//----------------------------------------------------------------------------//
// More step action in the list can be inserted here, upto ab is tested:      //
//----------------------------------------------------------------------------//
r007: NOP   0; //Wrong action number
      S     #sqSequencer.Error_Fault;
      JU    k007; //Exit
_007: NOP   0; // Action error handling
      JU    k007; // Exit






NETWORK
TITLE =S007:: STEP-007:: : ACTION CODE
    //================================ ACT HEADER ============================//
    // ACTION ACTION ACTION ACTION ACTION ACTION ACTION ACTION ACTION ACTION  //
    // AUTOCODE   AUTOCODE   AUTOCODE   AUTOCODE   AUTOCODE   AUTOCODE   AUTO //
    // ACTION ACTION ACTION ACTION ACTION ACTION ACTION ACTION ACTION ACTION  //
    //------------------------------------------------------------------------//
    // //Open Mx steam supply on WFI/PS lines.
    // //
    // //Log steam opened time.
    aa07: NOP   0;

    //------------------------------------------------------------------------//
    // ACT ACT ACT ACT ACT ACT ACT ACT ACT ACT ACT ACT ACT ACT ACT ACT ACT    //
    //------------------------------------------------------------------------//
    //Set emc_water to substate FLUSH and open WFI/PS supply valve.
L "dbCONST".SEL.LIQUID.PSWFI;
T #_emc_water_medium_liquid;
L 0;
T #_emc_water_runtime;
L "dbCONST".BLK.EMC2.SUBS.FLUSH;
T #_emc_water_subs;
L "dbCONST".BLK.CMD.START;
T #_emc_water_cmd;


//Log steam opened time.
SET;
S #_log_msg_steam_open;

    //------------------------------------------------------------------------//
    // VERIFY  VERIFY VERIFY VERIFY VERIFY VERIFY VERIFY VERIFY VERIFY VERIFY //
    //------------------------------------------------------------------------//
    //Verify if emc_water changed to substate FLUSH.
A(;
L   #_emc_water_subs;
L   "dbCONST".BLK.EMC2.SUBS.FLUSH;
==I;
);
    S     #sqSequencer.STEP.ActionVerified; //Action verified

    //------------------------------------------------------------------------//
    // Action done:                                                           //
    //------------------------------------------------------------------------//
    O     #sqSequencer.STEP.ActionVerified;
    O     #smc.NO_VERIFIC;       //No verification , bypass verification code
    S     #sqSequencer.STEP.ActionFinished;






    //============================= STEP FOOTER ==============================//
    // AUTOCODE   AUTOCODE   AUTOCODE   AUTOCODE   AUTOCODE   AUTOCODE   AUTO //
    // Get Ready after action finished:                                       //
    //------------------------------------------------------------------------//
    A     #sqSequencer.STEP.ActionFinished;
    JCN   k007;

    //------------------------------------------------------------------------//
    // Reset Action finished flag, ready for next step action:                //
    //------------------------------------------------------------------------//
    R     #sqSequencer.STEP.ActionVerified;
    R     #sqSequencer.STEP.ActionFinished;

    //------------------------------------------------------------------------//
    // If ALL actions are finished:                                           //
    //------------------------------------------------------------------------//
    SET   ;
    S     #sqSequencer.STEP.Finished;
    R     #sqSequencer.STEP.Active;
    S     #sqSequencer.STEP.Done[07];

    //------------------------------------------------------------------------//
    // End Step action(s):                                                    //
    //------------------------------------------------------------------------//
    JU    k007;

//----------------------------------------------------------------------------//
// Finished Step Action(s):                                                   //
//----------------------------------------------------------------------------//
k007: NOP   0;

    A     #sqStepTimerExpired;
    S     #sqSequencer.STEP.WithError[07]; // Step error flag
    S     #sqSequencer.Error_Fault;
    R     #sqStepTimer.IN;

NETWORK
TITLE =S007:STEP-007::Begin Transition
    //------------------------------------------------------------------------//
    // Begin the transition code:                                             //
    //------------------------------------------------------------------------//
    A007: NOP   0;
    R     #sqStepTimer.IN;






    //============================= TRAN HEADER ==============================//
    // AUTOCODE   AUTOCODE   AUTOCODE   AUTOCODE   AUTOCODE   AUTOCODE   AUTO //
    // Bypass transition if manual jump:                                      //
    //------------------------------------------------------------------------//
    A     #sqSequencer.STEP.Finished;
    A     #smc.TRN_AND_JUMP;     //Manual jump is set Transition as bypassed
    JCN   COMM;              //exit

NETWORK
TITLE =S007::STEP 007:TRAN 009: Pressure check
//----------------------------------------------------------------------------//
// TRAN   TRAN   TRAN   TRAN   TRAN   TRAN   TRAN   TRAN   TRAN   TRAN   TRAN //
// TRAN   TRAN   TRAN   TRAN   TRAN   TRAN   TRAN   TRAN   TRAN   TRAN   TRAN //
//----------------------------------------------------------------------------//
// Pressure increased above PRES_STM_POS. PCx013> PRES_STM_POS
//----------------------------------------------------------------------------//
// CONDITION   CONDITION   CONDITION   CONDITION   CONDITION   CONDITION   CO //
// CONDITION   CONDITION   CONDITION   CONDITION   CONDITION   CONDITION   CO //
//----------------------------------------------------------------------------//
A(;
L 	#_emc_gas_pi_vessel_pv;
L 	#_r_pres_stm_pos;
>R;
);






    //============================= TRAN FOOTER ==============================//
    // Transition jump control:                                               //
    //------------------------------------------------------------------------//
    A     #sqSequencer.STEP.JumpCtrl;
    S     #sqSequencer.STEP.Jump;
    S     #sqSequencer.STEP.jumpDone[07];

NETWORK
TITLE =S007:t009::TRANS-v: EXIT TRANSITION AND READY THE NEXT STEP
    //------------------------------------------------------------------------//
    // Check the jump flag and jump to the next step if the transition        //
    // condition is true and has set the jump flag:                           //
    //------------------------------------------------------------------------//
    A     #sqSequencer.STEP.Jump;
    JCN   x009;

    R     #sqSequencer.STEP.Jump;
    R     #sqSequencer.STEP.Finished;

    L     08;     // Load next STEPNO to jump to if transition satisfied
    T     #sqSequencer.STEP.NumberNext; //Next Step08.

    JU    COMM;              // Transition satisfied, Exit, go to next step
x009: NOP   0;






NETWORK
TITLE =S007::STEP-007:EXIT TRANSITION:
    //========================== STEP TRANSFER ===============================//
    // Jump to the common step progression code:                              //
    //------------------------------------------------------------------------//
    JU    COMM;






NETWORK
TITLE =S008: STEP-08::UO_MX_SIP : Positive pressure.
    //================================ STEP HEADER ===========================//
    // STEP008 STEP008 STEP008 STEP008
    // AUTOCODE   AUTOCODE   AUTOCODE   AUTOCODE   AUTOCODE   AUTOCODE   AUTO //
    // STEP008 STEP008 STEP008 STEP008
    //------------------------------------------------------------------------//
    // Positive pressure has been achieved.
    // Log actual positive pressure.
    //
    // Open Mx SIP condensate drain valve and vent filter drain valve.
    //------------------------------------------------------------------------//
S008: NOP   0;

      SET;
      R     #sqSequencer.STEP.jumpDone[08];
      A     #sqSequencer.CMD.Pause; //If paused jump
      JC    COMM;

NETWORK
TITLE =S008:STEP-08:Begin Action

      A     #sqSequencer.STEP.Finished;
      JC    A008; // Exit Action code, Jump to A008 Transition code

      //----------------------------------------------------------------------//
      // Begin step Action:                                                   //
      //----------------------------------------------------------------------//
      A     #sqSequencer.STEP.Active;
      JC    L008; // Action number loaded, Jump to L008--Step Action List

      //----------------------------------------------------------------------//
      // Load Default/Initial Step action number:                             //
      //----------------------------------------------------------------------//
      S     #sqSequencer.STEP.Active;
      S     #sqStepTimer.IN;
      L     1; //First Action, Step must contain Minimum one action
      T     #sqSequencer.STEP.ActionNumber;

//----------------------------------------------------------------------------//
// Step action list.                                                          //
// aann=mini Action step number(aa) inside main step number(nn)               //
// First Action aa00, Second action ab00, Third ac00, etc.                    //
//----------------------------------------------------------------------------//
L008: NOP   0;

      L     #sqSequencer.STEP.ActionNumber;
      JL    r008; //Wrong Action number
      JU    _008; //Action error handling
       JU    aa08; //ACTION-01
JU    ab08; //ACTION-02


//----------------------------------------------------------------------------//
// More step action in the list can be inserted here, upto ab is tested:      //
//----------------------------------------------------------------------------//
r008: NOP   0; //Wrong action number
      S     #sqSequencer.Error_Fault;
      JU    k008; //Exit
_008: NOP   0; // Action error handling
      JU    k008; // Exit






NETWORK
TITLE =S008:: STEP-008:: : ACTION CODE
    //================================ ACT HEADER ============================//
    // ACTION ACTION ACTION ACTION ACTION ACTION ACTION ACTION ACTION ACTION  //
    // AUTOCODE   AUTOCODE   AUTOCODE   AUTOCODE   AUTOCODE   AUTOCODE   AUTO //
    // ACTION ACTION ACTION ACTION ACTION ACTION ACTION ACTION ACTION ACTION  //
    //------------------------------------------------------------------------//
    // //Log actual positive pressure.
    // //Open Mx SIP condensate drain valve and vent filter drain valve.
    aa08: NOP   0;

    //------------------------------------------------------------------------//
    // ACT ACT ACT ACT ACT ACT ACT ACT ACT ACT ACT ACT ACT ACT ACT ACT ACT    //
    //------------------------------------------------------------------------//
    //Log actual positive pressure.
L #_emc_gas_pi_vessel_pv;
T #_real_positive_pressure;

SET;
S #_log_real_positive_pressure;

//Start EMX4_SIP.
L "dbCONST".BLK.EMX4.SUBS.SIP;
T #_emx_drain_subs;
L "dbCONST".BLK.CMD.START;
T #_emx_drain_cmd;

// Set vessel VENT filter EM to substate SIP
L "dbCONST".BLK.EMG1.SUBS.SIP;
T #_emg_filter_subs;
L "dbCONST".BLK.CMD.START;
T #_emg_filter_cmd;

//Open gas line drain valve.
L "dbCONST".SEL.GAS.DRAIN;
T #_emc_gas_medium_gas;
L "dbCONST".BLK.CMD.RESTART;
T #_emc_gas_cmd;

    //------------------------------------------------------------------------//
    // VERIFY  VERIFY VERIFY VERIFY VERIFY VERIFY VERIFY VERIFY VERIFY VERIFY //
    //------------------------------------------------------------------------//
    A(;
L #_emx_drain_subs;
L "dbCONST".BLK.EMX4.SUBS.SIP;
==I;
);
A(;
L #_emg_filter_subs;
L "dbCONST".BLK.EMG1.SUBS.SIP;
==I;
);
A(;
L   #_emc_gas_state;
L   "dbCONST".BLK.STATE.STOPPED;
>I;
);
A(;
L   #_emc_gas_state;
L   "dbCONST".BLK.STATE.INTERLOCKED;
<I;
);

    S     #sqSequencer.STEP.ActionVerified; //Action verified

    //------------------------------------------------------------------------//
    // Action done:                                                           //
    //------------------------------------------------------------------------//
    O     #sqSequencer.STEP.ActionVerified;
    O     #smc.NO_VERIFIC;       //No verification , bypass verification code
    S     #sqSequencer.STEP.ActionFinished;






    //============================= ACT FOOTER ===============================//
    // AUTOCODE   AUTOCODE   AUTOCODE   AUTOCODE   AUTOCODE   AUTOCODE   AUTO //
    // Get Ready after action finished:                                       //
    //------------------------------------------------------------------------//
    A     #sqSequencer.STEP.ActionFinished;
    JCN   k008;

    //------------------------------------------------------------------------//
    // Reset Action finished flag, ready for next step action:                //
    //------------------------------------------------------------------------//
    R     #sqSequencer.STEP.ActionVerified;
    R     #sqSequencer.STEP.ActionFinished;

    //------------------------------------------------------------------------//
    // Load Next Step Action number:                                          //
    //------------------------------------------------------------------------//
    L     02; //Load next Action
    T     #sqSequencer.STEP.ActionNumber;






NETWORK
TITLE =S008:: STEP-008:: : ACTION CODE
    //================================ ACT HEADER ============================//
    // ACTION ACTION ACTION ACTION ACTION ACTION ACTION ACTION ACTION ACTION  //
    // AUTOCODE   AUTOCODE   AUTOCODE   AUTOCODE   AUTOCODE   AUTOCODE   AUTO //
    // ACTION ACTION ACTION ACTION ACTION ACTION ACTION ACTION ACTION ACTION  //
    //------------------------------------------------------------------------//
    // //Clear gas EM restart command
    ab08: NOP   0;

    //------------------------------------------------------------------------//
    // ACT ACT ACT ACT ACT ACT ACT ACT ACT ACT ACT ACT ACT ACT ACT ACT ACT    //
    //------------------------------------------------------------------------//
    L "dbCONST".BLK.CMD.START;
T #_emc_gas_cmd;

    //------------------------------------------------------------------------//
    // VERIFY  VERIFY VERIFY VERIFY VERIFY VERIFY VERIFY VERIFY VERIFY VERIFY //
    //------------------------------------------------------------------------//

    S     #sqSequencer.STEP.ActionVerified; //Action verified

    //------------------------------------------------------------------------//
    // Action done:                                                           //
    //------------------------------------------------------------------------//
    O     #sqSequencer.STEP.ActionVerified;
    O     #smc.NO_VERIFIC;       //No verification , bypass verification code
    S     #sqSequencer.STEP.ActionFinished;






    //============================= STEP FOOTER ==============================//
    // AUTOCODE   AUTOCODE   AUTOCODE   AUTOCODE   AUTOCODE   AUTOCODE   AUTO //
    // Get Ready after action finished:                                       //
    //------------------------------------------------------------------------//
    A     #sqSequencer.STEP.ActionFinished;
    JCN   k008;

    //------------------------------------------------------------------------//
    // Reset Action finished flag, ready for next step action:                //
    //------------------------------------------------------------------------//
    R     #sqSequencer.STEP.ActionVerified;
    R     #sqSequencer.STEP.ActionFinished;

    //------------------------------------------------------------------------//
    // If ALL actions are finished:                                           //
    //------------------------------------------------------------------------//
    SET   ;
    S     #sqSequencer.STEP.Finished;
    R     #sqSequencer.STEP.Active;
    S     #sqSequencer.STEP.Done[08];

    //------------------------------------------------------------------------//
    // End Step action(s):                                                    //
    //------------------------------------------------------------------------//
    JU    k008;

//----------------------------------------------------------------------------//
// Finished Step Action(s):                                                   //
//----------------------------------------------------------------------------//
k008: NOP   0;

    A     #sqStepTimerExpired;
    S     #sqSequencer.STEP.WithError[08]; // Step error flag
    S     #sqSequencer.Error_Fault;
    R     #sqStepTimer.IN;

NETWORK
TITLE =S008:STEP-008::Begin Transition
    //------------------------------------------------------------------------//
    // Begin the transition code:                                             //
    //------------------------------------------------------------------------//
    A008: NOP   0;
    R     #sqStepTimer.IN;






    //============================= TRAN HEADER ==============================//
    // AUTOCODE   AUTOCODE   AUTOCODE   AUTOCODE   AUTOCODE   AUTOCODE   AUTO //
    // Bypass transition if manual jump:                                      //
    //------------------------------------------------------------------------//
    A     #sqSequencer.STEP.Finished;
    A     #smc.TRN_AND_JUMP;     //Manual jump is set Transition as bypassed
    JCN   COMM;              //exit

NETWORK
TITLE =S008::STEP 008:TRAN 010: Empty Transition
//----------------------------------------------------------------------------//
// TRAN   TRAN   TRAN   TRAN   TRAN   TRAN   TRAN   TRAN   TRAN   TRAN   TRAN //
// TRAN   TRAN   TRAN   TRAN   TRAN   TRAN   TRAN   TRAN   TRAN   TRAN   TRAN //
//----------------------------------------------------------------------------//
// Empty Transition
//----------------------------------------------------------------------------//
// CONDITION   CONDITION   CONDITION   CONDITION   CONDITION   CONDITION   CO //
// CONDITION   CONDITION   CONDITION   CONDITION   CONDITION   CONDITION   CO //
//----------------------------------------------------------------------------//
A "uncondJump";






    //============================= TRAN FOOTER ==============================//
    // Transition jump control:                                               //
    //------------------------------------------------------------------------//
    A     #sqSequencer.STEP.JumpCtrl;
    S     #sqSequencer.STEP.Jump;
    S     #sqSequencer.STEP.jumpDone[08];

NETWORK
TITLE =S008:t010::TRANS-v: EXIT TRANSITION AND READY THE NEXT STEP
    //------------------------------------------------------------------------//
    // Check the jump flag and jump to the next step if the transition        //
    // condition is true and has set the jump flag:                           //
    //------------------------------------------------------------------------//
    A     #sqSequencer.STEP.Jump;
    JCN   x010;

    R     #sqSequencer.STEP.Jump;
    R     #sqSequencer.STEP.Finished;

    L     09;     // Load next STEPNO to jump to if transition satisfied
    T     #sqSequencer.STEP.NumberNext; //Next Step09.

    JU    COMM;              // Transition satisfied, Exit, go to next step
x010: NOP   0;






NETWORK
TITLE =S008::STEP-008:EXIT TRANSITION:
    //========================== STEP TRANSFER ===============================//
    // Jump to the common step progression code:                              //
    //------------------------------------------------------------------------//
    JU    COMM;






NETWORK
TITLE =S009: STEP-09::UO_MX_SIP : Wait for free steaming timer
    //================================ STEP HEADER ===========================//
    // STEP009 STEP009 STEP009 STEP009
    // AUTOCODE   AUTOCODE   AUTOCODE   AUTOCODE   AUTOCODE   AUTOCODE   AUTO //
    // STEP009 STEP009 STEP009 STEP009
    //------------------------------------------------------------------------//
    // Start timer TIME_STM_DRAIN_Mx
    //------------------------------------------------------------------------//
S009: NOP   0;

      SET;
      R     #sqSequencer.STEP.jumpDone[09];
      A     #sqSequencer.CMD.Pause; //If paused jump
      JC    COMM;

NETWORK
TITLE =S009:STEP-09:Begin Action

      A     #sqSequencer.STEP.Finished;
      JC    A009; // Exit Action code, Jump to A009 Transition code

      //----------------------------------------------------------------------//
      // Begin step Action:                                                   //
      //----------------------------------------------------------------------//
      A     #sqSequencer.STEP.Active;
      JC    L009; // Action number loaded, Jump to L009--Step Action List

      //----------------------------------------------------------------------//
      // Load Default/Initial Step action number:                             //
      //----------------------------------------------------------------------//
      S     #sqSequencer.STEP.Active;
      S     #sqStepTimer.IN;
      L     1; //First Action, Step must contain Minimum one action
      T     #sqSequencer.STEP.ActionNumber;

//----------------------------------------------------------------------------//
// Step action list.                                                          //
// aann=mini Action step number(aa) inside main step number(nn)               //
// First Action aa00, Second action ab00, Third ac00, etc.                    //
//----------------------------------------------------------------------------//
L009: NOP   0;

      L     #sqSequencer.STEP.ActionNumber;
      JL    r009; //Wrong Action number
      JU    _009; //Action error handling
       JU    aa09; //ACTION-01


//----------------------------------------------------------------------------//
// More step action in the list can be inserted here, upto ab is tested:      //
//----------------------------------------------------------------------------//
r009: NOP   0; //Wrong action number
      S     #sqSequencer.Error_Fault;
      JU    k009; //Exit
_009: NOP   0; // Action error handling
      JU    k009; // Exit






NETWORK
TITLE =S009:: STEP-009:: : ACTION CODE
    //================================ ACT HEADER ============================//
    // ACTION ACTION ACTION ACTION ACTION ACTION ACTION ACTION ACTION ACTION  //
    // AUTOCODE   AUTOCODE   AUTOCODE   AUTOCODE   AUTOCODE   AUTOCODE   AUTO //
    // ACTION ACTION ACTION ACTION ACTION ACTION ACTION ACTION ACTION ACTION  //
    //------------------------------------------------------------------------//
    // //Start timer TIME_STM_DRAIN_Mx
    aa09: NOP   0;

    //------------------------------------------------------------------------//
    // ACT ACT ACT ACT ACT ACT ACT ACT ACT ACT ACT ACT ACT ACT ACT ACT ACT    //
    //------------------------------------------------------------------------//
    //Start Timer for steaming
A #SQ_TIMER.Q;
R #sqSeqTimerStart;

AN #SQ_TIMER.Q;
S #sqSeqTimerStart;
L #_r_time_stm_drain_mx;
L 1000;
*I;
T #SQ_TIMER.PT;

    //------------------------------------------------------------------------//
    // VERIFY  VERIFY VERIFY VERIFY VERIFY VERIFY VERIFY VERIFY VERIFY VERIFY //
    //------------------------------------------------------------------------//
    A #sqSeqTimerStart;
    S     #sqSequencer.STEP.ActionVerified; //Action verified

    //------------------------------------------------------------------------//
    // Action done:                                                           //
    //------------------------------------------------------------------------//
    O     #sqSequencer.STEP.ActionVerified;
    O     #smc.NO_VERIFIC;       //No verification , bypass verification code
    S     #sqSequencer.STEP.ActionFinished;






    //============================= STEP FOOTER ==============================//
    // AUTOCODE   AUTOCODE   AUTOCODE   AUTOCODE   AUTOCODE   AUTOCODE   AUTO //
    // Get Ready after action finished:                                       //
    //------------------------------------------------------------------------//
    A     #sqSequencer.STEP.ActionFinished;
    JCN   k009;

    //------------------------------------------------------------------------//
    // Reset Action finished flag, ready for next step action:                //
    //------------------------------------------------------------------------//
    R     #sqSequencer.STEP.ActionVerified;
    R     #sqSequencer.STEP.ActionFinished;

    //------------------------------------------------------------------------//
    // If ALL actions are finished:                                           //
    //------------------------------------------------------------------------//
    SET   ;
    S     #sqSequencer.STEP.Finished;
    R     #sqSequencer.STEP.Active;
    S     #sqSequencer.STEP.Done[09];

    //------------------------------------------------------------------------//
    // End Step action(s):                                                    //
    //------------------------------------------------------------------------//
    JU    k009;

//----------------------------------------------------------------------------//
// Finished Step Action(s):                                                   //
//----------------------------------------------------------------------------//
k009: NOP   0;

    A     #sqStepTimerExpired;
    S     #sqSequencer.STEP.WithError[09]; // Step error flag
    S     #sqSequencer.Error_Fault;
    R     #sqStepTimer.IN;

NETWORK
TITLE =S009:STEP-009::Begin Transition
    //------------------------------------------------------------------------//
    // Begin the transition code:                                             //
    //------------------------------------------------------------------------//
    A009: NOP   0;
    R     #sqStepTimer.IN;






    //============================= TRAN HEADER ==============================//
    // AUTOCODE   AUTOCODE   AUTOCODE   AUTOCODE   AUTOCODE   AUTOCODE   AUTO //
    // Bypass transition if manual jump:                                      //
    //------------------------------------------------------------------------//
    A     #sqSequencer.STEP.Finished;
    A     #smc.TRN_AND_JUMP;     //Manual jump is set Transition as bypassed
    JCN   COMM;              //exit

NETWORK
TITLE =S009::STEP 009:TRAN 011: Timer expired
//----------------------------------------------------------------------------//
// TRAN   TRAN   TRAN   TRAN   TRAN   TRAN   TRAN   TRAN   TRAN   TRAN   TRAN //
// TRAN   TRAN   TRAN   TRAN   TRAN   TRAN   TRAN   TRAN   TRAN   TRAN   TRAN //
//----------------------------------------------------------------------------//
// Timer TIME_STM_DRAIN_Mx expired?
//----------------------------------------------------------------------------//
// CONDITION   CONDITION   CONDITION   CONDITION   CONDITION   CONDITION   CO //
// CONDITION   CONDITION   CONDITION   CONDITION   CONDITION   CONDITION   CO //
//----------------------------------------------------------------------------//
A #SQ_TIMER.Q;






    //============================= TRAN FOOTER ==============================//
    // Transition jump control:                                               //
    //------------------------------------------------------------------------//
    A     #sqSequencer.STEP.JumpCtrl;
    S     #sqSequencer.STEP.Jump;
    S     #sqSequencer.STEP.jumpDone[09];

NETWORK
TITLE =S009:t011::TRANS-v: EXIT TRANSITION AND READY THE NEXT STEP
    //------------------------------------------------------------------------//
    // Check the jump flag and jump to the next step if the transition        //
    // condition is true and has set the jump flag:                           //
    //------------------------------------------------------------------------//
    A     #sqSequencer.STEP.Jump;
    JCN   x011;

    R     #sqSequencer.STEP.Jump;
    R     #sqSequencer.STEP.Finished;

    L     10;     // Load next STEPNO to jump to if transition satisfied
    T     #sqSequencer.STEP.NumberNext; //Next Step10.

    JU    COMM;              // Transition satisfied, Exit, go to next step
x011: NOP   0;






NETWORK
TITLE =S009::STEP-009:EXIT TRANSITION:
    //========================== STEP TRANSFER ===============================//
    // Jump to the common step progression code:                              //
    //------------------------------------------------------------------------//
    JU    COMM;






NETWORK
TITLE =S010: STEP-10::UO_MX_SIP : Free steam complete.
    //================================ STEP HEADER ===========================//
    // STEP010 STEP010 STEP010 STEP010
    // AUTOCODE   AUTOCODE   AUTOCODE   AUTOCODE   AUTOCODE   AUTOCODE   AUTO //
    // STEP010 STEP010 STEP010 STEP010
    //------------------------------------------------------------------------//
    // Log closed system steaming start time
    //------------------------------------------------------------------------//
S010: NOP   0;

      SET;
      R     #sqSequencer.STEP.jumpDone[10];
      A     #sqSequencer.CMD.Pause; //If paused jump
      JC    COMM;

NETWORK
TITLE =S010:STEP-10:Begin Action

      A     #sqSequencer.STEP.Finished;
      JC    A010; // Exit Action code, Jump to A010 Transition code

      //----------------------------------------------------------------------//
      // Begin step Action:                                                   //
      //----------------------------------------------------------------------//
      A     #sqSequencer.STEP.Active;
      JC    L010; // Action number loaded, Jump to L010--Step Action List

      //----------------------------------------------------------------------//
      // Load Default/Initial Step action number:                             //
      //----------------------------------------------------------------------//
      S     #sqSequencer.STEP.Active;
      S     #sqStepTimer.IN;
      L     1; //First Action, Step must contain Minimum one action
      T     #sqSequencer.STEP.ActionNumber;

//----------------------------------------------------------------------------//
// Step action list.                                                          //
// aann=mini Action step number(aa) inside main step number(nn)               //
// First Action aa00, Second action ab00, Third ac00, etc.                    //
//----------------------------------------------------------------------------//
L010: NOP   0;

      L     #sqSequencer.STEP.ActionNumber;
      JL    r010; //Wrong Action number
      JU    _010; //Action error handling
       JU    aa10; //ACTION-01
JU    ab10; //ACTION-02


//----------------------------------------------------------------------------//
// More step action in the list can be inserted here, upto ab is tested:      //
//----------------------------------------------------------------------------//
r010: NOP   0; //Wrong action number
      S     #sqSequencer.Error_Fault;
      JU    k010; //Exit
_010: NOP   0; // Action error handling
      JU    k010; // Exit






NETWORK
TITLE =S010:: STEP-010:: : ACTION CODE
    //================================ ACT HEADER ============================//
    // ACTION ACTION ACTION ACTION ACTION ACTION ACTION ACTION ACTION ACTION  //
    // AUTOCODE   AUTOCODE   AUTOCODE   AUTOCODE   AUTOCODE   AUTOCODE   AUTO //
    // ACTION ACTION ACTION ACTION ACTION ACTION ACTION ACTION ACTION ACTION  //
    //------------------------------------------------------------------------//
    // //Stop MMFLx to reset it
    aa10: NOP   0;

    //------------------------------------------------------------------------//
    // ACT ACT ACT ACT ACT ACT ACT ACT ACT ACT ACT ACT ACT ACT ACT ACT ACT    //
    //------------------------------------------------------------------------//
    L "dbCONST".BLK.CMD.STOP;
T #_emx_mmfl_cmd;

    //------------------------------------------------------------------------//
    // VERIFY  VERIFY VERIFY VERIFY VERIFY VERIFY VERIFY VERIFY VERIFY VERIFY //
    //------------------------------------------------------------------------//
    A(;
L   #_emx_mmfl_state;
L   "dbCONST".BLK.STATE.STOPPED;
==I;
);
    S     #sqSequencer.STEP.ActionVerified; //Action verified

    //------------------------------------------------------------------------//
    // Action done:                                                           //
    //------------------------------------------------------------------------//
    O     #sqSequencer.STEP.ActionVerified;
    O     #smc.NO_VERIFIC;       //No verification , bypass verification code
    S     #sqSequencer.STEP.ActionFinished;






    //============================= ACT FOOTER ===============================//
    // AUTOCODE   AUTOCODE   AUTOCODE   AUTOCODE   AUTOCODE   AUTOCODE   AUTO //
    // Get Ready after action finished:                                       //
    //------------------------------------------------------------------------//
    A     #sqSequencer.STEP.ActionFinished;
    JCN   k010;

    //------------------------------------------------------------------------//
    // Reset Action finished flag, ready for next step action:                //
    //------------------------------------------------------------------------//
    R     #sqSequencer.STEP.ActionVerified;
    R     #sqSequencer.STEP.ActionFinished;

    //------------------------------------------------------------------------//
    // Load Next Step Action number:                                          //
    //------------------------------------------------------------------------//
    L     02; //Load next Action
    T     #sqSequencer.STEP.ActionNumber;






NETWORK
TITLE =S010:: STEP-010:: : ACTION CODE
    //================================ ACT HEADER ============================//
    // ACTION ACTION ACTION ACTION ACTION ACTION ACTION ACTION ACTION ACTION  //
    // AUTOCODE   AUTOCODE   AUTOCODE   AUTOCODE   AUTOCODE   AUTOCODE   AUTO //
    // ACTION ACTION ACTION ACTION ACTION ACTION ACTION ACTION ACTION ACTION  //
    //------------------------------------------------------------------------//
    // //Log closed system start time
    // //Start pulsing MMFLx valves
    ab10: NOP   0;

    //------------------------------------------------------------------------//
    // ACT ACT ACT ACT ACT ACT ACT ACT ACT ACT ACT ACT ACT ACT ACT ACT ACT    //
    //------------------------------------------------------------------------//
    //Log closed system start time.
SET;
S #_log_msg_steam_closed;

// Set emx_mmfl to substate SIP_PULSE and start it.
L _r_time_mmflx_pulse_heat;
L 1000;
*I;
T #_emx_mmfl_opened_time;
L "dbCONST".BLK.EMX1.SUBS.SIP_PULSE;
T #_emx_mmfl_subs;
L "dbCONST".BLK.CMD.START;
T #_emx_mmfl_cmd;

    //------------------------------------------------------------------------//
    // VERIFY  VERIFY VERIFY VERIFY VERIFY VERIFY VERIFY VERIFY VERIFY VERIFY //
    //------------------------------------------------------------------------//

    S     #sqSequencer.STEP.ActionVerified; //Action verified

    //------------------------------------------------------------------------//
    // Action done:                                                           //
    //------------------------------------------------------------------------//
    O     #sqSequencer.STEP.ActionVerified;
    O     #smc.NO_VERIFIC;       //No verification , bypass verification code
    S     #sqSequencer.STEP.ActionFinished;






    //============================= STEP FOOTER ==============================//
    // AUTOCODE   AUTOCODE   AUTOCODE   AUTOCODE   AUTOCODE   AUTOCODE   AUTO //
    // Get Ready after action finished:                                       //
    //------------------------------------------------------------------------//
    A     #sqSequencer.STEP.ActionFinished;
    JCN   k010;

    //------------------------------------------------------------------------//
    // Reset Action finished flag, ready for next step action:                //
    //------------------------------------------------------------------------//
    R     #sqSequencer.STEP.ActionVerified;
    R     #sqSequencer.STEP.ActionFinished;

    //------------------------------------------------------------------------//
    // If ALL actions are finished:                                           //
    //------------------------------------------------------------------------//
    SET   ;
    S     #sqSequencer.STEP.Finished;
    R     #sqSequencer.STEP.Active;
    S     #sqSequencer.STEP.Done[10];

    //------------------------------------------------------------------------//
    // End Step action(s):                                                    //
    //------------------------------------------------------------------------//
    JU    k010;

//----------------------------------------------------------------------------//
// Finished Step Action(s):                                                   //
//----------------------------------------------------------------------------//
k010: NOP   0;

    A     #sqStepTimerExpired;
    S     #sqSequencer.STEP.WithError[10]; // Step error flag
    S     #sqSequencer.Error_Fault;
    R     #sqStepTimer.IN;

NETWORK
TITLE =S010:STEP-010::Begin Transition
    //------------------------------------------------------------------------//
    // Begin the transition code:                                             //
    //------------------------------------------------------------------------//
    A010: NOP   0;
    R     #sqStepTimer.IN;






    //============================= TRAN HEADER ==============================//
    // AUTOCODE   AUTOCODE   AUTOCODE   AUTOCODE   AUTOCODE   AUTOCODE   AUTO //
    // Bypass transition if manual jump:                                      //
    //------------------------------------------------------------------------//
    A     #sqSequencer.STEP.Finished;
    A     #smc.TRN_AND_JUMP;     //Manual jump is set Transition as bypassed
    JCN   COMM;              //exit

NETWORK
TITLE =S010::STEP 010:TRAN 012: Empty Transition
//----------------------------------------------------------------------------//
// TRAN   TRAN   TRAN   TRAN   TRAN   TRAN   TRAN   TRAN   TRAN   TRAN   TRAN //
// TRAN   TRAN   TRAN   TRAN   TRAN   TRAN   TRAN   TRAN   TRAN   TRAN   TRAN //
//----------------------------------------------------------------------------//
// Empty Transition
//----------------------------------------------------------------------------//
// CONDITION   CONDITION   CONDITION   CONDITION   CONDITION   CONDITION   CO //
// CONDITION   CONDITION   CONDITION   CONDITION   CONDITION   CONDITION   CO //
//----------------------------------------------------------------------------//
A "uncondJump";






    //============================= TRAN FOOTER ==============================//
    // Transition jump control:                                               //
    //------------------------------------------------------------------------//
    A     #sqSequencer.STEP.JumpCtrl;
    S     #sqSequencer.STEP.Jump;
    S     #sqSequencer.STEP.jumpDone[10];

NETWORK
TITLE =S010:t012::TRANS-v: EXIT TRANSITION AND READY THE NEXT STEP
    //------------------------------------------------------------------------//
    // Check the jump flag and jump to the next step if the transition        //
    // condition is true and has set the jump flag:                           //
    //------------------------------------------------------------------------//
    A     #sqSequencer.STEP.Jump;
    JCN   x012;

    R     #sqSequencer.STEP.Jump;
    R     #sqSequencer.STEP.Finished;

    L     11;     // Load next STEPNO to jump to if transition satisfied
    T     #sqSequencer.STEP.NumberNext; //Next Step11.

    JU    COMM;              // Transition satisfied, Exit, go to next step
x012: NOP   0;






NETWORK
TITLE =S010::STEP-010:EXIT TRANSITION:
    //========================== STEP TRANSFER ===============================//
    // Jump to the common step progression code:                              //
    //------------------------------------------------------------------------//
    JU    COMM;






NETWORK
TITLE =S011: STEP-11::UO_MX_SIP : SIP Started
    //================================ STEP HEADER ===========================//
    // STEP011 STEP011 STEP011 STEP011
    // AUTOCODE   AUTOCODE   AUTOCODE   AUTOCODE   AUTOCODE   AUTOCODE   AUTO //
    // STEP011 STEP011 STEP011 STEP011
    //------------------------------------------------------------------------//
    // Skip timer for SIP_ABORT if sip_timer_started=FALSE.
    //------------------------------------------------------------------------//
S011: NOP   0;

      SET;
      R     #sqSequencer.STEP.jumpDone[11];
      A     #sqSequencer.CMD.Pause; //If paused jump
      JC    COMM;

NETWORK
TITLE =S011:STEP-11:Begin Action

      A     #sqSequencer.STEP.Finished;
      JC    A011; // Exit Action code, Jump to A011 Transition code

      //----------------------------------------------------------------------//
      // Begin step Action:                                                   //
      //----------------------------------------------------------------------//
      A     #sqSequencer.STEP.Active;
      JC    L011; // Action number loaded, Jump to L011--Step Action List

      //----------------------------------------------------------------------//
      // Load Default/Initial Step action number:                             //
      //----------------------------------------------------------------------//
      S     #sqSequencer.STEP.Active;
      S     #sqStepTimer.IN;
      L     1; //First Action, Step must contain Minimum one action
      T     #sqSequencer.STEP.ActionNumber;

//----------------------------------------------------------------------------//
// Step action list.                                                          //
// aann=mini Action step number(aa) inside main step number(nn)               //
// First Action aa00, Second action ab00, Third ac00, etc.                    //
//----------------------------------------------------------------------------//
L011: NOP   0;

      L     #sqSequencer.STEP.ActionNumber;
      JL    r011; //Wrong Action number
      JU    _011; //Action error handling
       JU    aa11; //ACTION-01


//----------------------------------------------------------------------------//
// More step action in the list can be inserted here, upto ab is tested:      //
//----------------------------------------------------------------------------//
r011: NOP   0; //Wrong action number
      S     #sqSequencer.Error_Fault;
      JU    k011; //Exit
_011: NOP   0; // Action error handling
      JU    k011; // Exit






NETWORK
TITLE =S011:: STEP-011:: : ACTION CODE
    //================================ ACT HEADER ============================//
    // ACTION ACTION ACTION ACTION ACTION ACTION ACTION ACTION ACTION ACTION  //
    // AUTOCODE   AUTOCODE   AUTOCODE   AUTOCODE   AUTOCODE   AUTOCODE   AUTO //
    // ACTION ACTION ACTION ACTION ACTION ACTION ACTION ACTION ACTION ACTION  //
    //------------------------------------------------------------------------//
    // //Skip timer for SIP_ABORT if sip_timer_started=FALSE.
    aa11: NOP   0;

    //------------------------------------------------------------------------//
    // ACT ACT ACT ACT ACT ACT ACT ACT ACT ACT ACT ACT ACT ACT ACT ACT ACT    //
    //------------------------------------------------------------------------//
    //Skip timer for SIP_ABORT if sip_timer_started=FALSE.
A #_sip_timer_started;
JC tsi1;

// Start SIP ABORT timer
A #SQ_TIMER3.Q;
R #sqSeqTimerStart3;

AN #SQ_TIMER3.Q;
S #sqSeqTimerStart3;
L #_r_time_sip_abort;
L 1000;
*I;
T #SQ_TIMER3.PT;


tsi1: NOP 0;
//SIP started.


    //------------------------------------------------------------------------//
    // VERIFY  VERIFY VERIFY VERIFY VERIFY VERIFY VERIFY VERIFY VERIFY VERIFY //
    //------------------------------------------------------------------------//
    A "uncondJump";
    S     #sqSequencer.STEP.ActionVerified; //Action verified

    //------------------------------------------------------------------------//
    // Action done:                                                           //
    //------------------------------------------------------------------------//
    O     #sqSequencer.STEP.ActionVerified;
    O     #smc.NO_VERIFIC;       //No verification , bypass verification code
    S     #sqSequencer.STEP.ActionFinished;






    //============================= STEP FOOTER ==============================//
    // AUTOCODE   AUTOCODE   AUTOCODE   AUTOCODE   AUTOCODE   AUTOCODE   AUTO //
    // Get Ready after action finished:                                       //
    //------------------------------------------------------------------------//
    A     #sqSequencer.STEP.ActionFinished;
    JCN   k011;

    //------------------------------------------------------------------------//
    // Reset Action finished flag, ready for next step action:                //
    //------------------------------------------------------------------------//
    R     #sqSequencer.STEP.ActionVerified;
    R     #sqSequencer.STEP.ActionFinished;

    //------------------------------------------------------------------------//
    // If ALL actions are finished:                                           //
    //------------------------------------------------------------------------//
    SET   ;
    S     #sqSequencer.STEP.Finished;
    R     #sqSequencer.STEP.Active;
    S     #sqSequencer.STEP.Done[11];

    //------------------------------------------------------------------------//
    // End Step action(s):                                                    //
    //------------------------------------------------------------------------//
    JU    k011;

//----------------------------------------------------------------------------//
// Finished Step Action(s):                                                   //
//----------------------------------------------------------------------------//
k011: NOP   0;

    A     #sqStepTimerExpired;
    S     #sqSequencer.STEP.WithError[11]; // Step error flag
    S     #sqSequencer.Error_Fault;
    R     #sqStepTimer.IN;

NETWORK
TITLE =S011:STEP-011::Begin Transition
    //------------------------------------------------------------------------//
    // Begin the transition code:                                             //
    //------------------------------------------------------------------------//
    A011: NOP   0;
    R     #sqStepTimer.IN;






    //============================= TRAN HEADER ==============================//
    // AUTOCODE   AUTOCODE   AUTOCODE   AUTOCODE   AUTOCODE   AUTOCODE   AUTO //
    // Bypass transition if manual jump:                                      //
    //------------------------------------------------------------------------//
    A     #sqSequencer.STEP.Finished;
    A     #smc.TRN_AND_JUMP;     //Manual jump is set Transition as bypassed
    JCN   COMM;              //exit

NETWORK
TITLE =S011::STEP 011:TRAN 013: Empty Transition
//----------------------------------------------------------------------------//
// TRAN   TRAN   TRAN   TRAN   TRAN   TRAN   TRAN   TRAN   TRAN   TRAN   TRAN //
// TRAN   TRAN   TRAN   TRAN   TRAN   TRAN   TRAN   TRAN   TRAN   TRAN   TRAN //
//----------------------------------------------------------------------------//
// Empty Transition
//----------------------------------------------------------------------------//
// CONDITION   CONDITION   CONDITION   CONDITION   CONDITION   CONDITION   CO //
// CONDITION   CONDITION   CONDITION   CONDITION   CONDITION   CONDITION   CO //
//----------------------------------------------------------------------------//
A "uncondJump";






    //============================= TRAN FOOTER ==============================//
    // Transition jump control:                                               //
    //------------------------------------------------------------------------//
    A     #sqSequencer.STEP.JumpCtrl;
    S     #sqSequencer.STEP.Jump;
    S     #sqSequencer.STEP.jumpDone[11];

NETWORK
TITLE =S011:t013::TRANS-v: EXIT TRANSITION AND READY THE NEXT STEP
    //------------------------------------------------------------------------//
    // Check the jump flag and jump to the next step if the transition        //
    // condition is true and has set the jump flag:                           //
    //------------------------------------------------------------------------//
    A     #sqSequencer.STEP.Jump;
    JCN   x013;

    R     #sqSequencer.STEP.Jump;
    R     #sqSequencer.STEP.Finished;

    L     12;     // Load next STEPNO to jump to if transition satisfied
    T     #sqSequencer.STEP.NumberNext; //Next Step12.

    JU    COMM;              // Transition satisfied, Exit, go to next step
x013: NOP   0;






NETWORK
TITLE =S011::STEP-011:EXIT TRANSITION:
    //========================== STEP TRANSFER ===============================//
    // Jump to the common step progression code:                              //
    //------------------------------------------------------------------------//
    JU    COMM;






NETWORK
TITLE =S012: STEP-12::UO_MX_SIP : Mixing Vessel SIP
    //================================ STEP HEADER ===========================//
    // STEP012 STEP012 STEP012 STEP012
    // AUTOCODE   AUTOCODE   AUTOCODE   AUTOCODE   AUTOCODE   AUTOCODE   AUTO //
    // STEP012 STEP012 STEP012 STEP012
    //------------------------------------------------------------------------//
    // Reset log message flags
    //------------------------------------------------------------------------//
S012: NOP   0;

      SET;
      R     #sqSequencer.STEP.jumpDone[12];
      A     #sqSequencer.CMD.Pause; //If paused jump
      JC    COMM;

NETWORK
TITLE =S012:STEP-12:Begin Action

      A     #sqSequencer.STEP.Finished;
      JC    A012; // Exit Action code, Jump to A012 Transition code

      //----------------------------------------------------------------------//
      // Begin step Action:                                                   //
      //----------------------------------------------------------------------//
      A     #sqSequencer.STEP.Active;
      JC    L012; // Action number loaded, Jump to L012--Step Action List

      //----------------------------------------------------------------------//
      // Load Default/Initial Step action number:                             //
      //----------------------------------------------------------------------//
      S     #sqSequencer.STEP.Active;
      S     #sqStepTimer.IN;
      L     1; //First Action, Step must contain Minimum one action
      T     #sqSequencer.STEP.ActionNumber;

//----------------------------------------------------------------------------//
// Step action list.                                                          //
// aann=mini Action step number(aa) inside main step number(nn)               //
// First Action aa00, Second action ab00, Third ac00, etc.                    //
//----------------------------------------------------------------------------//
L012: NOP   0;

      L     #sqSequencer.STEP.ActionNumber;
      JL    r012; //Wrong Action number
      JU    _012; //Action error handling
       JU    aa12; //ACTION-01


//----------------------------------------------------------------------------//
// More step action in the list can be inserted here, upto ab is tested:      //
//----------------------------------------------------------------------------//
r012: NOP   0; //Wrong action number
      S     #sqSequencer.Error_Fault;
      JU    k012; //Exit
_012: NOP   0; // Action error handling
      JU    k012; // Exit






NETWORK
TITLE =S012:: STEP-012:: : ACTION CODE
    //================================ ACT HEADER ============================//
    // ACTION ACTION ACTION ACTION ACTION ACTION ACTION ACTION ACTION ACTION  //
    // AUTOCODE   AUTOCODE   AUTOCODE   AUTOCODE   AUTOCODE   AUTOCODE   AUTO //
    // ACTION ACTION ACTION ACTION ACTION ACTION ACTION ACTION ACTION ACTION  //
    //------------------------------------------------------------------------//
    // //Reset message log flags
    aa12: NOP   0;

    //------------------------------------------------------------------------//
    // ACT ACT ACT ACT ACT ACT ACT ACT ACT ACT ACT ACT ACT ACT ACT ACT ACT    //
    //------------------------------------------------------------------------//
    SET;
R #_log_real_emt_ti_hex_pv;
R #_log_real_emg_ti_drain_pv;
R #_log_real_emv_ti_vessel_pv;
R #_log_real_emx_ti_drain_pv;

R #sqSeqTimerStart2;

AN #SQ_TIMER2.Q;
S #sqSeqTimerStart2;
L T#10S;
T #SQ_TIMER2.PT;

    //------------------------------------------------------------------------//
    // VERIFY  VERIFY VERIFY VERIFY VERIFY VERIFY VERIFY VERIFY VERIFY VERIFY //
    //------------------------------------------------------------------------//

    S     #sqSequencer.STEP.ActionVerified; //Action verified

    //------------------------------------------------------------------------//
    // Action done:                                                           //
    //------------------------------------------------------------------------//
    O     #sqSequencer.STEP.ActionVerified;
    O     #smc.NO_VERIFIC;       //No verification , bypass verification code
    S     #sqSequencer.STEP.ActionFinished;






    //============================= STEP FOOTER ==============================//
    // AUTOCODE   AUTOCODE   AUTOCODE   AUTOCODE   AUTOCODE   AUTOCODE   AUTO //
    // Get Ready after action finished:                                       //
    //------------------------------------------------------------------------//
    A     #sqSequencer.STEP.ActionFinished;
    JCN   k012;

    //------------------------------------------------------------------------//
    // Reset Action finished flag, ready for next step action:                //
    //------------------------------------------------------------------------//
    R     #sqSequencer.STEP.ActionVerified;
    R     #sqSequencer.STEP.ActionFinished;

    //------------------------------------------------------------------------//
    // If ALL actions are finished:                                           //
    //------------------------------------------------------------------------//
    SET   ;
    S     #sqSequencer.STEP.Finished;
    R     #sqSequencer.STEP.Active;
    S     #sqSequencer.STEP.Done[12];

    //------------------------------------------------------------------------//
    // End Step action(s):                                                    //
    //------------------------------------------------------------------------//
    JU    k012;

//----------------------------------------------------------------------------//
// Finished Step Action(s):                                                   //
//----------------------------------------------------------------------------//
k012: NOP   0;

    A     #sqStepTimerExpired;
    S     #sqSequencer.STEP.WithError[12]; // Step error flag
    S     #sqSequencer.Error_Fault;
    R     #sqStepTimer.IN;

NETWORK
TITLE =S012:STEP-012::Begin Transition
    //------------------------------------------------------------------------//
    // Begin the transition code:                                             //
    //------------------------------------------------------------------------//
    A012: NOP   0;
    R     #sqStepTimer.IN;






    //============================= TRAN HEADER ==============================//
    // AUTOCODE   AUTOCODE   AUTOCODE   AUTOCODE   AUTOCODE   AUTOCODE   AUTO //
    // Bypass transition if manual jump:                                      //
    //------------------------------------------------------------------------//
    A     #sqSequencer.STEP.Finished;
    A     #smc.TRN_AND_JUMP;     //Manual jump is set Transition as bypassed
    JCN   COMM;              //exit

NETWORK
TITLE =S012::STEP 012:TRAN 014: 10 seconds expired
//----------------------------------------------------------------------------//
// TRAN   TRAN   TRAN   TRAN   TRAN   TRAN   TRAN   TRAN   TRAN   TRAN   TRAN //
// TRAN   TRAN   TRAN   TRAN   TRAN   TRAN   TRAN   TRAN   TRAN   TRAN   TRAN //
//----------------------------------------------------------------------------//
// Jump after flags have had a chance to reset on HMI
//----------------------------------------------------------------------------//
// CONDITION   CONDITION   CONDITION   CONDITION   CONDITION   CONDITION   CO //
// CONDITION   CONDITION   CONDITION   CONDITION   CONDITION   CONDITION   CO //
//----------------------------------------------------------------------------//
A #SQ_TIMER2.Q;






    //============================= TRAN FOOTER ==============================//
    // Transition jump control:                                               //
    //------------------------------------------------------------------------//
    A     #sqSequencer.STEP.JumpCtrl;
    S     #sqSequencer.STEP.Jump;
    S     #sqSequencer.STEP.jumpDone[12];

NETWORK
TITLE =S012:t014::TRANS-v: EXIT TRANSITION AND READY THE NEXT STEP
    //------------------------------------------------------------------------//
    // Check the jump flag and jump to the next step if the transition        //
    // condition is true and has set the jump flag:                           //
    //------------------------------------------------------------------------//
    A     #sqSequencer.STEP.Jump;
    JCN   x014;

    R     #sqSequencer.STEP.Jump;
    R     #sqSequencer.STEP.Finished;

    L     13;     // Load next STEPNO to jump to if transition satisfied
    T     #sqSequencer.STEP.NumberNext; //Next Step13.

    JU    COMM;              // Transition satisfied, Exit, go to next step
x014: NOP   0;






NETWORK
TITLE =S012::STEP-012:EXIT TRANSITION:
    //========================== STEP TRANSFER ===============================//
    // Jump to the common step progression code:                              //
    //------------------------------------------------------------------------//
    JU    COMM;






NETWORK
TITLE =S013: STEP-13::UO_MX_SIP : Monitor MX SIP Temperatures
    //================================ STEP HEADER ===========================//
    // STEP013 STEP013 STEP013 STEP013
    // AUTOCODE   AUTOCODE   AUTOCODE   AUTOCODE   AUTOCODE   AUTOCODE   AUTO //
    // STEP013 STEP013 STEP013 STEP013
    //------------------------------------------------------------------------//
    // Log all Mx vessel temperatures every 30sec.
    //------------------------------------------------------------------------//
S013: NOP   0;

      SET;
      R     #sqSequencer.STEP.jumpDone[13];
      A     #sqSequencer.CMD.Pause; //If paused jump
      JC    COMM;

NETWORK
TITLE =S013:STEP-13:Begin Action

      A     #sqSequencer.STEP.Finished;
      JC    A013; // Exit Action code, Jump to A013 Transition code

      //----------------------------------------------------------------------//
      // Begin step Action:                                                   //
      //----------------------------------------------------------------------//
      A     #sqSequencer.STEP.Active;
      JC    L013; // Action number loaded, Jump to L013--Step Action List

      //----------------------------------------------------------------------//
      // Load Default/Initial Step action number:                             //
      //----------------------------------------------------------------------//
      S     #sqSequencer.STEP.Active;
      S     #sqStepTimer.IN;
      L     1; //First Action, Step must contain Minimum one action
      T     #sqSequencer.STEP.ActionNumber;

//----------------------------------------------------------------------------//
// Step action list.                                                          //
// aann=mini Action step number(aa) inside main step number(nn)               //
// First Action aa00, Second action ab00, Third ac00, etc.                    //
//----------------------------------------------------------------------------//
L013: NOP   0;

      L     #sqSequencer.STEP.ActionNumber;
      JL    r013; //Wrong Action number
      JU    _013; //Action error handling
       JU    aa13; //ACTION-01


//----------------------------------------------------------------------------//
// More step action in the list can be inserted here, upto ab is tested:      //
//----------------------------------------------------------------------------//
r013: NOP   0; //Wrong action number
      S     #sqSequencer.Error_Fault;
      JU    k013; //Exit
_013: NOP   0; // Action error handling
      JU    k013; // Exit






NETWORK
TITLE =S013:: STEP-013:: : ACTION CODE
    //================================ ACT HEADER ============================//
    // ACTION ACTION ACTION ACTION ACTION ACTION ACTION ACTION ACTION ACTION  //
    // AUTOCODE   AUTOCODE   AUTOCODE   AUTOCODE   AUTOCODE   AUTOCODE   AUTO //
    // ACTION ACTION ACTION ACTION ACTION ACTION ACTION ACTION ACTION ACTION  //
    //------------------------------------------------------------------------//
    // //Log all Mx vessel temperatures  every 30sec.
    aa13: NOP   0;

    //------------------------------------------------------------------------//
    // ACT ACT ACT ACT ACT ACT ACT ACT ACT ACT ACT ACT ACT ACT ACT ACT ACT    //
    //------------------------------------------------------------------------//
    //Log all temperatures
SET;
R #sqSeqTimerStart2;
L #_emt_hex_ti_hex_pv;
T #_real_emt_ti_hex_pv;
L #_emg_filter_ti_drain_pv;
T #_real_emg_ti_drain_pv;
L #_emv_vessel_ti_vessel_pv;
T #_real_emv_ti_vessel_pv;
L #_emx_drain_ti_drain_pv;
T #_real_emx_ti_drain_pv;

SET;
S #_log_real_emt_ti_hex_pv;
S #_log_real_emg_ti_drain_pv;
S #_log_real_emv_ti_vessel_pv;
S #_log_real_emx_ti_drain_pv;


AN #SQ_TIMER2.Q;
S #sqSeqTimerStart2;
L T#20S;
T #SQ_TIMER2.PT;

    //------------------------------------------------------------------------//
    // VERIFY  VERIFY VERIFY VERIFY VERIFY VERIFY VERIFY VERIFY VERIFY VERIFY //
    //------------------------------------------------------------------------//
    A "uncondJump";
    S     #sqSequencer.STEP.ActionVerified; //Action verified

    //------------------------------------------------------------------------//
    // Action done:                                                           //
    //------------------------------------------------------------------------//
    O     #sqSequencer.STEP.ActionVerified;
    O     #smc.NO_VERIFIC;       //No verification , bypass verification code
    S     #sqSequencer.STEP.ActionFinished;






    //============================= STEP FOOTER ==============================//
    // AUTOCODE   AUTOCODE   AUTOCODE   AUTOCODE   AUTOCODE   AUTOCODE   AUTO //
    // Get Ready after action finished:                                       //
    //------------------------------------------------------------------------//
    A     #sqSequencer.STEP.ActionFinished;
    JCN   k013;

    //------------------------------------------------------------------------//
    // Reset Action finished flag, ready for next step action:                //
    //------------------------------------------------------------------------//
    R     #sqSequencer.STEP.ActionVerified;
    R     #sqSequencer.STEP.ActionFinished;

    //------------------------------------------------------------------------//
    // If ALL actions are finished:                                           //
    //------------------------------------------------------------------------//
    SET   ;
    S     #sqSequencer.STEP.Finished;
    R     #sqSequencer.STEP.Active;
    S     #sqSequencer.STEP.Done[13];

    //------------------------------------------------------------------------//
    // End Step action(s):                                                    //
    //------------------------------------------------------------------------//
    JU    k013;

//----------------------------------------------------------------------------//
// Finished Step Action(s):                                                   //
//----------------------------------------------------------------------------//
k013: NOP   0;

    A     #sqStepTimerExpired;
    S     #sqSequencer.STEP.WithError[13]; // Step error flag
    S     #sqSequencer.Error_Fault;
    R     #sqStepTimer.IN;

NETWORK
TITLE =S013:STEP-013::Begin Transition
    //------------------------------------------------------------------------//
    // Begin the transition code:                                             //
    //------------------------------------------------------------------------//
    A013: NOP   0;
    R     #sqStepTimer.IN;






    //============================= TRAN HEADER ==============================//
    // AUTOCODE   AUTOCODE   AUTOCODE   AUTOCODE   AUTOCODE   AUTOCODE   AUTO //
    // Bypass transition if manual jump:                                      //
    //------------------------------------------------------------------------//
    A     #sqSequencer.STEP.Finished;
    A     #smc.TRN_AND_JUMP;     //Manual jump is set Transition as bypassed
    JCN   COMM;              //exit

NETWORK
TITLE =S013::STEP 013:TRAN 015: Temperature below setpoint
//----------------------------------------------------------------------------//
// TRAN   TRAN   TRAN   TRAN   TRAN   TRAN   TRAN   TRAN   TRAN   TRAN   TRAN //
// TRAN   TRAN   TRAN   TRAN   TRAN   TRAN   TRAN   TRAN   TRAN   TRAN   TRAN //
//----------------------------------------------------------------------------//
// SIP timer running and any temperature below TEMP_SIP or the vent filter inlet temperature below TEMP_SIP_VENT?
//----------------------------------------------------------------------------//
// CONDITION   CONDITION   CONDITION   CONDITION   CONDITION   CONDITION   CO //
// CONDITION   CONDITION   CONDITION   CONDITION   CONDITION   CONDITION   CO //
//----------------------------------------------------------------------------//
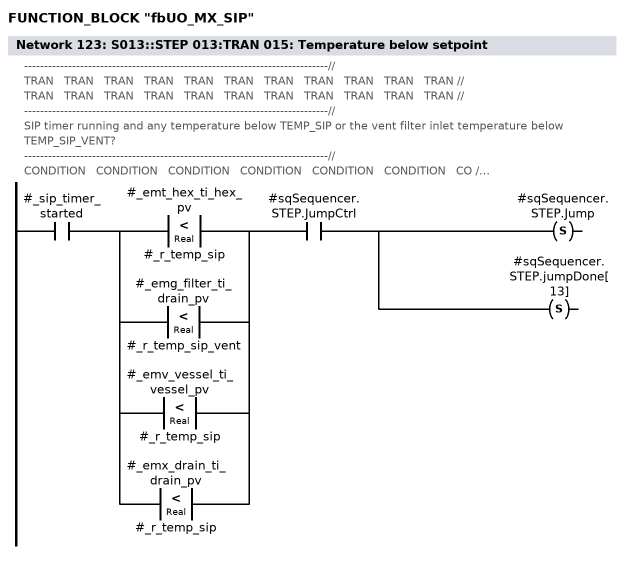
A #_sip_timer_started;
A(;
//TIn109
O(;
L 	#_emt_hex_ti_hex_pv;
L 	#_r_temp_sip;
<R;
);
//TIn103
O(;
L              #_emg_filter_ti_drain_pv;
L 	#_r_temp_sip_vent;
<R;
);
//TIn105
O(;
L              #_emv_vessel_ti_vessel_pv;
L 	#_r_temp_sip;
<R;
);
//TIn107.
O(;
L              #_emx_drain_ti_drain_pv;
L 	#_r_temp_sip;
<R;
);
);






    //============================= TRAN FOOTER ==============================//
    // Transition jump control:                                               //
    //------------------------------------------------------------------------//
    A     #sqSequencer.STEP.JumpCtrl;
    S     #sqSequencer.STEP.Jump;
    S     #sqSequencer.STEP.jumpDone[13];

NETWORK
TITLE =S013:t015::TRANS-v: EXIT TRANSITION AND READY THE NEXT STEP
    //------------------------------------------------------------------------//
    // Check the jump flag and jump to the next step if the transition        //
    // condition is true and has set the jump flag:                           //
    //------------------------------------------------------------------------//
    A     #sqSequencer.STEP.Jump;
    JCN   x015;

    R     #sqSequencer.STEP.Jump;
    R     #sqSequencer.STEP.Finished;

    L     15;     // Load next STEPNO to jump to if transition satisfied
    T     #sqSequencer.STEP.NumberNext; //Next Step15.

    JU    COMM;              // Transition satisfied, Exit, go to next step
x015: NOP   0;






    //============================= TRAN HEADER ==============================//
    // AUTOCODE   AUTOCODE   AUTOCODE   AUTOCODE   AUTOCODE   AUTOCODE   AUTO //
    // Bypass transition if manual jump:                                      //
    //------------------------------------------------------------------------//
    A     #sqSequencer.STEP.Finished;
    A     #smc.TRN_AND_JUMP;     //Manual jump is set Transition as bypassed
    JCN   COMM;              //exit

NETWORK
TITLE =S013::STEP 013:TRAN 016: All temperatures above setpoint.
//----------------------------------------------------------------------------//
// TRAN   TRAN   TRAN   TRAN   TRAN   TRAN   TRAN   TRAN   TRAN   TRAN   TRAN //
// TRAN   TRAN   TRAN   TRAN   TRAN   TRAN   TRAN   TRAN   TRAN   TRAN   TRAN //
//----------------------------------------------------------------------------//
// All SIP temperatures above TEMP_SIP °C and the vent filter inlet temperature above TEMP_SIP_VENT?
    // and SIP timer not running?
    // Mx HEX Outlet TI_x109, Mx vent line TI_x103, Mx Vessel TI_x105, MFLx Filtration Line TI_x107 & Mx Drain TI_x109.
//----------------------------------------------------------------------------//
// CONDITION   CONDITION   CONDITION   CONDITION   CONDITION   CONDITION   CO //
// CONDITION   CONDITION   CONDITION   CONDITION   CONDITION   CONDITION   CO //
//----------------------------------------------------------------------------//
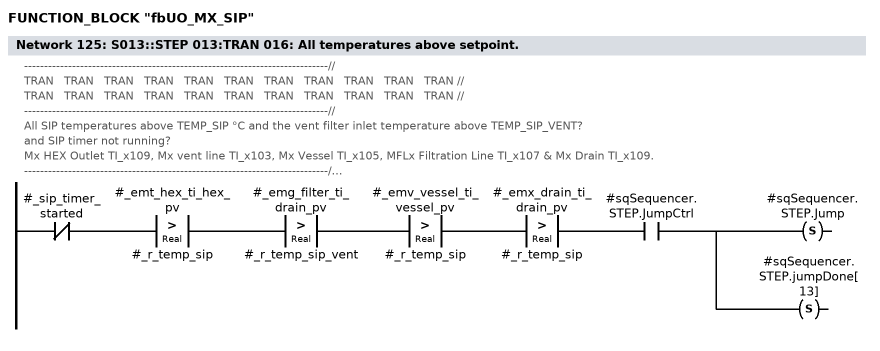
AN #_sip_timer_started;

//TIn109
A(;
L 	#_emt_hex_ti_hex_pv;
L 	#_r_temp_sip;
>R;
);
//TIn103
A(;
L              #_emg_filter_ti_drain_pv;
L 	#_r_temp_sip_vent;
>R;
);
//TIn105
A(;
L              #_emv_vessel_ti_vessel_pv;
L 	#_r_temp_sip;
>R;
);
//TIn107.
A(;
L              #_emx_drain_ti_drain_pv;
L 	#_r_temp_sip;
>R;
);






    //============================= TRAN FOOTER ==============================//
    // Transition jump control:                                               //
    //------------------------------------------------------------------------//
    A     #sqSequencer.STEP.JumpCtrl;
    S     #sqSequencer.STEP.Jump;
    S     #sqSequencer.STEP.jumpDone[13];

NETWORK
TITLE =S013:t016::TRANS-v: EXIT TRANSITION AND READY THE NEXT STEP
    //------------------------------------------------------------------------//
    // Check the jump flag and jump to the next step if the transition        //
    // condition is true and has set the jump flag:                           //
    //------------------------------------------------------------------------//
    A     #sqSequencer.STEP.Jump;
    JCN   x016;

    R     #sqSequencer.STEP.Jump;
    R     #sqSequencer.STEP.Finished;

    L     14;     // Load next STEPNO to jump to if transition satisfied
    T     #sqSequencer.STEP.NumberNext; //Next Step14.

    JU    COMM;              // Transition satisfied, Exit, go to next step
x016: NOP   0;






    //============================= TRAN HEADER ==============================//
    // AUTOCODE   AUTOCODE   AUTOCODE   AUTOCODE   AUTOCODE   AUTOCODE   AUTO //
    // Bypass transition if manual jump:                                      //
    //------------------------------------------------------------------------//
    A     #sqSequencer.STEP.Finished;
    A     #smc.TRN_AND_JUMP;     //Manual jump is set Transition as bypassed
    JCN   COMM;              //exit

NETWORK
TITLE =S013::STEP 013:TRAN 017: Temperature logging timer expired
//----------------------------------------------------------------------------//
// TRAN   TRAN   TRAN   TRAN   TRAN   TRAN   TRAN   TRAN   TRAN   TRAN   TRAN //
// TRAN   TRAN   TRAN   TRAN   TRAN   TRAN   TRAN   TRAN   TRAN   TRAN   TRAN //
//----------------------------------------------------------------------------//
// 20 seconds expired.
//----------------------------------------------------------------------------//
// CONDITION   CONDITION   CONDITION   CONDITION   CONDITION   CONDITION   CO //
// CONDITION   CONDITION   CONDITION   CONDITION   CONDITION   CONDITION   CO //
//----------------------------------------------------------------------------//
A #SQ_TIMER2.Q;






    //============================= TRAN FOOTER ==============================//
    // Transition jump control:                                               //
    //------------------------------------------------------------------------//
    A     #sqSequencer.STEP.JumpCtrl;
    S     #sqSequencer.STEP.Jump;
    S     #sqSequencer.STEP.jumpDone[13];

NETWORK
TITLE =S013:t017::TRANS-v: EXIT TRANSITION AND READY THE NEXT STEP
    //------------------------------------------------------------------------//
    // Check the jump flag and jump to the next step if the transition        //
    // condition is true and has set the jump flag:                           //
    //------------------------------------------------------------------------//
    A     #sqSequencer.STEP.Jump;
    JCN   x017;

    R     #sqSequencer.STEP.Jump;
    R     #sqSequencer.STEP.Finished;

    L     12;     // Load next STEPNO to jump to if transition satisfied
    T     #sqSequencer.STEP.NumberNext; //Next Step12.

    JU    COMM;              // Transition satisfied, Exit, go to next step
x017: NOP   0;






    //============================= TRAN HEADER ==============================//
    // AUTOCODE   AUTOCODE   AUTOCODE   AUTOCODE   AUTOCODE   AUTOCODE   AUTO //
    // Bypass transition if manual jump:                                      //
    //------------------------------------------------------------------------//
    A     #sqSequencer.STEP.Finished;
    A     #smc.TRN_AND_JUMP;     //Manual jump is set Transition as bypassed
    JCN   COMM;              //exit

NETWORK
TITLE =S013::STEP 013:TRAN 018: SIP Timer Expired
//----------------------------------------------------------------------------//
// TRAN   TRAN   TRAN   TRAN   TRAN   TRAN   TRAN   TRAN   TRAN   TRAN   TRAN //
// TRAN   TRAN   TRAN   TRAN   TRAN   TRAN   TRAN   TRAN   TRAN   TRAN   TRAN //
//----------------------------------------------------------------------------//
// Timer TIME_SIP expired.
//----------------------------------------------------------------------------//
// CONDITION   CONDITION   CONDITION   CONDITION   CONDITION   CONDITION   CO //
// CONDITION   CONDITION   CONDITION   CONDITION   CONDITION   CONDITION   CO //
//----------------------------------------------------------------------------//
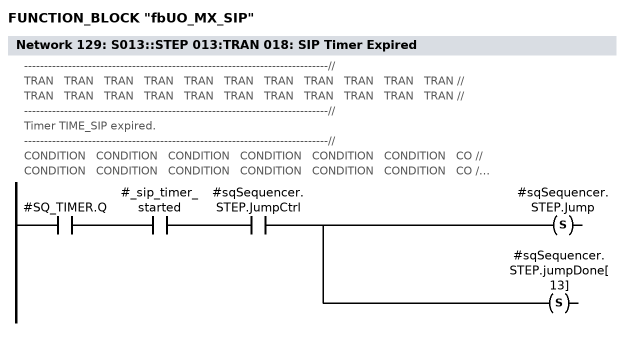
A #SQ_TIMER.Q;
A #_sip_timer_started;






    //============================= TRAN FOOTER ==============================//
    // Transition jump control:                                               //
    //------------------------------------------------------------------------//
    A     #sqSequencer.STEP.JumpCtrl;
    S     #sqSequencer.STEP.Jump;
    S     #sqSequencer.STEP.jumpDone[13];

NETWORK
TITLE =S013:t018::TRANS-v: EXIT TRANSITION AND READY THE NEXT STEP
    //------------------------------------------------------------------------//
    // Check the jump flag and jump to the next step if the transition        //
    // condition is true and has set the jump flag:                           //
    //------------------------------------------------------------------------//
    A     #sqSequencer.STEP.Jump;
    JCN   x018;

    R     #sqSequencer.STEP.Jump;
    R     #sqSequencer.STEP.Finished;

    L     16;     // Load next STEPNO to jump to if transition satisfied
    T     #sqSequencer.STEP.NumberNext; //Next Step16.

    JU    COMM;              // Transition satisfied, Exit, go to next step
x018: NOP   0;






    //============================= TRAN HEADER ==============================//
    // AUTOCODE   AUTOCODE   AUTOCODE   AUTOCODE   AUTOCODE   AUTOCODE   AUTO //
    // Bypass transition if manual jump:                                      //
    //------------------------------------------------------------------------//
    A     #sqSequencer.STEP.Finished;
    A     #smc.TRN_AND_JUMP;     //Manual jump is set Transition as bypassed
    JCN   COMM;              //exit

NETWORK
TITLE =S013::STEP 013:TRAN 019: Abort timer expired
//----------------------------------------------------------------------------//
// TRAN   TRAN   TRAN   TRAN   TRAN   TRAN   TRAN   TRAN   TRAN   TRAN   TRAN //
// TRAN   TRAN   TRAN   TRAN   TRAN   TRAN   TRAN   TRAN   TRAN   TRAN   TRAN //
//----------------------------------------------------------------------------//
// Timer TIME_SIP_ABORT is expired.
//----------------------------------------------------------------------------//
// CONDITION   CONDITION   CONDITION   CONDITION   CONDITION   CONDITION   CO //
// CONDITION   CONDITION   CONDITION   CONDITION   CONDITION   CONDITION   CO //
//----------------------------------------------------------------------------//
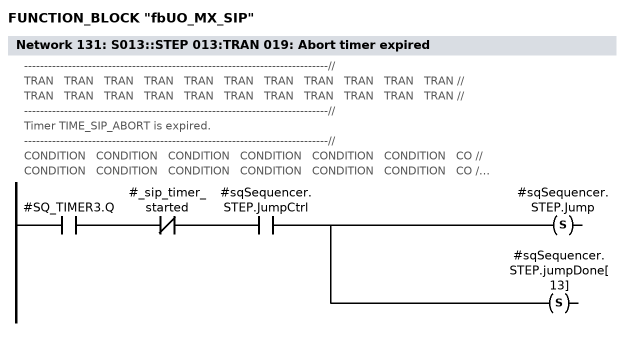
A #SQ_TIMER3.Q;
AN #_sip_timer_started;






    //============================= TRAN FOOTER ==============================//
    // Transition jump control:                                               //
    //------------------------------------------------------------------------//
    A     #sqSequencer.STEP.JumpCtrl;
    S     #sqSequencer.STEP.Jump;
    S     #sqSequencer.STEP.jumpDone[13];

NETWORK
TITLE =S013:t019::TRANS-v: EXIT TRANSITION AND READY THE NEXT STEP
    //------------------------------------------------------------------------//
    // Check the jump flag and jump to the next step if the transition        //
    // condition is true and has set the jump flag:                           //
    //------------------------------------------------------------------------//
    A     #sqSequencer.STEP.Jump;
    JCN   x019;

    R     #sqSequencer.STEP.Jump;
    R     #sqSequencer.STEP.Finished;

    L     17;     // Load next STEPNO to jump to if transition satisfied
    T     #sqSequencer.STEP.NumberNext; //Next Step17.

    JU    COMM;              // Transition satisfied, Exit, go to next step
x019: NOP   0;






NETWORK
TITLE =S013::STEP-013:EXIT TRANSITION:
    //========================== STEP TRANSFER ===============================//
    // Jump to the common step progression code:                              //
    //------------------------------------------------------------------------//
    JU    COMM;






NETWORK
TITLE =S014: STEP-14::UO_MX_SIP : Start MX SIP timer
    //================================ STEP HEADER ===========================//
    // STEP014 STEP014 STEP014 STEP014
    // AUTOCODE   AUTOCODE   AUTOCODE   AUTOCODE   AUTOCODE   AUTOCODE   AUTO //
    // STEP014 STEP014 STEP014 STEP014
    //------------------------------------------------------------------------//
    // Start SIP timer TIME_SIP.
    // Set sip_timer_started.
    // Log SIP start time.
    //------------------------------------------------------------------------//
S014: NOP   0;

      SET;
      R     #sqSequencer.STEP.jumpDone[14];
      A     #sqSequencer.CMD.Pause; //If paused jump
      JC    COMM;

NETWORK
TITLE =S014:STEP-14:Begin Action

      A     #sqSequencer.STEP.Finished;
      JC    A014; // Exit Action code, Jump to A014 Transition code

      //----------------------------------------------------------------------//
      // Begin step Action:                                                   //
      //----------------------------------------------------------------------//
      A     #sqSequencer.STEP.Active;
      JC    L014; // Action number loaded, Jump to L014--Step Action List

      //----------------------------------------------------------------------//
      // Load Default/Initial Step action number:                             //
      //----------------------------------------------------------------------//
      S     #sqSequencer.STEP.Active;
      S     #sqStepTimer.IN;
      L     1; //First Action, Step must contain Minimum one action
      T     #sqSequencer.STEP.ActionNumber;

//----------------------------------------------------------------------------//
// Step action list.                                                          //
// aann=mini Action step number(aa) inside main step number(nn)               //
// First Action aa00, Second action ab00, Third ac00, etc.                    //
//----------------------------------------------------------------------------//
L014: NOP   0;

      L     #sqSequencer.STEP.ActionNumber;
      JL    r014; //Wrong Action number
      JU    _014; //Action error handling
       JU    aa14; //ACTION-01


//----------------------------------------------------------------------------//
// More step action in the list can be inserted here, upto ab is tested:      //
//----------------------------------------------------------------------------//
r014: NOP   0; //Wrong action number
      S     #sqSequencer.Error_Fault;
      JU    k014; //Exit
_014: NOP   0; // Action error handling
      JU    k014; // Exit






NETWORK
TITLE =S014:: STEP-014:: : ACTION CODE
    //================================ ACT HEADER ============================//
    // ACTION ACTION ACTION ACTION ACTION ACTION ACTION ACTION ACTION ACTION  //
    // AUTOCODE   AUTOCODE   AUTOCODE   AUTOCODE   AUTOCODE   AUTOCODE   AUTO //
    // ACTION ACTION ACTION ACTION ACTION ACTION ACTION ACTION ACTION ACTION  //
    //------------------------------------------------------------------------//
    // //Start SIP timer TIME_SIP.
    // //Log SIP start time and Set sip_timer_started.
    aa14: NOP   0;

    //------------------------------------------------------------------------//
    // ACT ACT ACT ACT ACT ACT ACT ACT ACT ACT ACT ACT ACT ACT ACT ACT ACT    //
    //------------------------------------------------------------------------//
    A #SQ_TIMER.Q;
R #sqSeqTimerStart;

AN #SQ_TIMER.Q;
S #sqSeqTimerStart;
L #_r_time_sip;
L 1000;
*I;
T #SQ_TIMER.PT;

//Log SIP start time.
SET;
S #_log_msg_sip_start;
//SIP timer started
S #_sip_timer_started;

// Update emx_mmfl pulse time
L _r_time_mmflx_pulse_sip;
L 1000;
*I;
T #_emx_mmfl_opened_time;

    //------------------------------------------------------------------------//
    // VERIFY  VERIFY VERIFY VERIFY VERIFY VERIFY VERIFY VERIFY VERIFY VERIFY //
    //------------------------------------------------------------------------//
    A #sqSeqTimerStart;
    S     #sqSequencer.STEP.ActionVerified; //Action verified

    //------------------------------------------------------------------------//
    // Action done:                                                           //
    //------------------------------------------------------------------------//
    O     #sqSequencer.STEP.ActionVerified;
    O     #smc.NO_VERIFIC;       //No verification , bypass verification code
    S     #sqSequencer.STEP.ActionFinished;






    //============================= STEP FOOTER ==============================//
    // AUTOCODE   AUTOCODE   AUTOCODE   AUTOCODE   AUTOCODE   AUTOCODE   AUTO //
    // Get Ready after action finished:                                       //
    //------------------------------------------------------------------------//
    A     #sqSequencer.STEP.ActionFinished;
    JCN   k014;

    //------------------------------------------------------------------------//
    // Reset Action finished flag, ready for next step action:                //
    //------------------------------------------------------------------------//
    R     #sqSequencer.STEP.ActionVerified;
    R     #sqSequencer.STEP.ActionFinished;

    //------------------------------------------------------------------------//
    // If ALL actions are finished:                                           //
    //------------------------------------------------------------------------//
    SET   ;
    S     #sqSequencer.STEP.Finished;
    R     #sqSequencer.STEP.Active;
    S     #sqSequencer.STEP.Done[14];

    //------------------------------------------------------------------------//
    // End Step action(s):                                                    //
    //------------------------------------------------------------------------//
    JU    k014;

//----------------------------------------------------------------------------//
// Finished Step Action(s):                                                   //
//----------------------------------------------------------------------------//
k014: NOP   0;

    A     #sqStepTimerExpired;
    S     #sqSequencer.STEP.WithError[14]; // Step error flag
    S     #sqSequencer.Error_Fault;
    R     #sqStepTimer.IN;

NETWORK
TITLE =S014:STEP-014::Begin Transition
    //------------------------------------------------------------------------//
    // Begin the transition code:                                             //
    //------------------------------------------------------------------------//
    A014: NOP   0;
    R     #sqStepTimer.IN;






    //============================= TRAN HEADER ==============================//
    // AUTOCODE   AUTOCODE   AUTOCODE   AUTOCODE   AUTOCODE   AUTOCODE   AUTO //
    // Bypass transition if manual jump:                                      //
    //------------------------------------------------------------------------//
    A     #sqSequencer.STEP.Finished;
    A     #smc.TRN_AND_JUMP;     //Manual jump is set Transition as bypassed
    JCN   COMM;              //exit

NETWORK
TITLE =S014::STEP 014:TRAN 020: SIP Timer Expired
//----------------------------------------------------------------------------//
// TRAN   TRAN   TRAN   TRAN   TRAN   TRAN   TRAN   TRAN   TRAN   TRAN   TRAN //
// TRAN   TRAN   TRAN   TRAN   TRAN   TRAN   TRAN   TRAN   TRAN   TRAN   TRAN //
//----------------------------------------------------------------------------//
// Timer TIME_SIP not yet expired.
//----------------------------------------------------------------------------//
// CONDITION   CONDITION   CONDITION   CONDITION   CONDITION   CONDITION   CO //
// CONDITION   CONDITION   CONDITION   CONDITION   CONDITION   CONDITION   CO //
//----------------------------------------------------------------------------//
AN #SQ_TIMER.Q;






    //============================= TRAN FOOTER ==============================//
    // Transition jump control:                                               //
    //------------------------------------------------------------------------//
    A     #sqSequencer.STEP.JumpCtrl;
    S     #sqSequencer.STEP.Jump;
    S     #sqSequencer.STEP.jumpDone[14];

NETWORK
TITLE =S014:t020::TRANS-v: EXIT TRANSITION AND READY THE NEXT STEP
    //------------------------------------------------------------------------//
    // Check the jump flag and jump to the next step if the transition        //
    // condition is true and has set the jump flag:                           //
    //------------------------------------------------------------------------//
    A     #sqSequencer.STEP.Jump;
    JCN   x020;

    R     #sqSequencer.STEP.Jump;
    R     #sqSequencer.STEP.Finished;

    L     11;     // Load next STEPNO to jump to if transition satisfied
    T     #sqSequencer.STEP.NumberNext; //Next Step11.

    JU    COMM;              // Transition satisfied, Exit, go to next step
x020: NOP   0;






NETWORK
TITLE =S014::STEP-014:EXIT TRANSITION:
    //========================== STEP TRANSFER ===============================//
    // Jump to the common step progression code:                              //
    //------------------------------------------------------------------------//
    JU    COMM;






NETWORK
TITLE =S015: STEP-15::UO_MX_SIP : Low MX temperature during SIP
    //================================ STEP HEADER ===========================//
    // STEP015 STEP015 STEP015 STEP015
    // AUTOCODE   AUTOCODE   AUTOCODE   AUTOCODE   AUTOCODE   AUTOCODE   AUTO //
    // STEP015 STEP015 STEP015 STEP015
    //------------------------------------------------------------------------//
    // Reset sip_timer_started and log timer RESET.
    // Increase counter.
    //------------------------------------------------------------------------//
S015: NOP   0;

      SET;
      R     #sqSequencer.STEP.jumpDone[15];
      A     #sqSequencer.CMD.Pause; //If paused jump
      JC    COMM;

NETWORK
TITLE =S015:STEP-15:Begin Action

      A     #sqSequencer.STEP.Finished;
      JC    A015; // Exit Action code, Jump to A015 Transition code

      //----------------------------------------------------------------------//
      // Begin step Action:                                                   //
      //----------------------------------------------------------------------//
      A     #sqSequencer.STEP.Active;
      JC    L015; // Action number loaded, Jump to L015--Step Action List

      //----------------------------------------------------------------------//
      // Load Default/Initial Step action number:                             //
      //----------------------------------------------------------------------//
      S     #sqSequencer.STEP.Active;
      S     #sqStepTimer.IN;
      L     1; //First Action, Step must contain Minimum one action
      T     #sqSequencer.STEP.ActionNumber;

//----------------------------------------------------------------------------//
// Step action list.                                                          //
// aann=mini Action step number(aa) inside main step number(nn)               //
// First Action aa00, Second action ab00, Third ac00, etc.                    //
//----------------------------------------------------------------------------//
L015: NOP   0;

      L     #sqSequencer.STEP.ActionNumber;
      JL    r015; //Wrong Action number
      JU    _015; //Action error handling
       JU    aa15; //ACTION-01


//----------------------------------------------------------------------------//
// More step action in the list can be inserted here, upto ab is tested:      //
//----------------------------------------------------------------------------//
r015: NOP   0; //Wrong action number
      S     #sqSequencer.Error_Fault;
      JU    k015; //Exit
_015: NOP   0; // Action error handling
      JU    k015; // Exit






NETWORK
TITLE =S015:: STEP-015:: : ACTION CODE
    //================================ ACT HEADER ============================//
    // ACTION ACTION ACTION ACTION ACTION ACTION ACTION ACTION ACTION ACTION  //
    // AUTOCODE   AUTOCODE   AUTOCODE   AUTOCODE   AUTOCODE   AUTOCODE   AUTO //
    // ACTION ACTION ACTION ACTION ACTION ACTION ACTION ACTION ACTION ACTION  //
    //------------------------------------------------------------------------//
    // //Reset sip_timer_started and log timer RESET.
    // //Increase counter.
    aa15: NOP   0;

    //------------------------------------------------------------------------//
    // ACT ACT ACT ACT ACT ACT ACT ACT ACT ACT ACT ACT ACT ACT ACT ACT ACT    //
    //------------------------------------------------------------------------//
    A #SQ_TIMER.Q;
R #sqSeqTimerStart;

//Reset flag.
SET;
R #_sip_timer_started;
S #_log_msg_sip_timer_reset;

//Increase counter.
L #_ctr_sip_abort;
INC 1;
T #_ctr_sip_abort;

    //------------------------------------------------------------------------//
    // VERIFY  VERIFY VERIFY VERIFY VERIFY VERIFY VERIFY VERIFY VERIFY VERIFY //
    //------------------------------------------------------------------------//
    A "uncondJump";
    S     #sqSequencer.STEP.ActionVerified; //Action verified

    //------------------------------------------------------------------------//
    // Action done:                                                           //
    //------------------------------------------------------------------------//
    O     #sqSequencer.STEP.ActionVerified;
    O     #smc.NO_VERIFIC;       //No verification , bypass verification code
    S     #sqSequencer.STEP.ActionFinished;






    //============================= STEP FOOTER ==============================//
    // AUTOCODE   AUTOCODE   AUTOCODE   AUTOCODE   AUTOCODE   AUTOCODE   AUTO //
    // Get Ready after action finished:                                       //
    //------------------------------------------------------------------------//
    A     #sqSequencer.STEP.ActionFinished;
    JCN   k015;

    //------------------------------------------------------------------------//
    // Reset Action finished flag, ready for next step action:                //
    //------------------------------------------------------------------------//
    R     #sqSequencer.STEP.ActionVerified;
    R     #sqSequencer.STEP.ActionFinished;

    //------------------------------------------------------------------------//
    // If ALL actions are finished:                                           //
    //------------------------------------------------------------------------//
    SET   ;
    S     #sqSequencer.STEP.Finished;
    R     #sqSequencer.STEP.Active;
    S     #sqSequencer.STEP.Done[15];

    //------------------------------------------------------------------------//
    // End Step action(s):                                                    //
    //------------------------------------------------------------------------//
    JU    k015;

//----------------------------------------------------------------------------//
// Finished Step Action(s):                                                   //
//----------------------------------------------------------------------------//
k015: NOP   0;

    A     #sqStepTimerExpired;
    S     #sqSequencer.STEP.WithError[15]; // Step error flag
    S     #sqSequencer.Error_Fault;
    R     #sqStepTimer.IN;

NETWORK
TITLE =S015:STEP-015::Begin Transition
    //------------------------------------------------------------------------//
    // Begin the transition code:                                             //
    //------------------------------------------------------------------------//
    A015: NOP   0;
    R     #sqStepTimer.IN;






    //============================= TRAN HEADER ==============================//
    // AUTOCODE   AUTOCODE   AUTOCODE   AUTOCODE   AUTOCODE   AUTOCODE   AUTO //
    // Bypass transition if manual jump:                                      //
    //------------------------------------------------------------------------//
    A     #sqSequencer.STEP.Finished;
    A     #smc.TRN_AND_JUMP;     //Manual jump is set Transition as bypassed
    JCN   COMM;              //exit

NETWORK
TITLE =S015::STEP 015:TRAN 021: Retry SIP again
//----------------------------------------------------------------------------//
// TRAN   TRAN   TRAN   TRAN   TRAN   TRAN   TRAN   TRAN   TRAN   TRAN   TRAN //
// TRAN   TRAN   TRAN   TRAN   TRAN   TRAN   TRAN   TRAN   TRAN   TRAN   TRAN //
//----------------------------------------------------------------------------//
// Temperature has dropped less than 'NUM_SIP_ABORT' times
//----------------------------------------------------------------------------//
// CONDITION   CONDITION   CONDITION   CONDITION   CONDITION   CONDITION   CO //
// CONDITION   CONDITION   CONDITION   CONDITION   CONDITION   CONDITION   CO //
//----------------------------------------------------------------------------//
A(;
L 	#_ctr_sip_abort;
L 	#_r_num_sip_abort;
<I;
);






    //============================= TRAN FOOTER ==============================//
    // Transition jump control:                                               //
    //------------------------------------------------------------------------//
    A     #sqSequencer.STEP.JumpCtrl;
    S     #sqSequencer.STEP.Jump;
    S     #sqSequencer.STEP.jumpDone[15];

NETWORK
TITLE =S015:t021::TRANS-v: EXIT TRANSITION AND READY THE NEXT STEP
    //------------------------------------------------------------------------//
    // Check the jump flag and jump to the next step if the transition        //
    // condition is true and has set the jump flag:                           //
    //------------------------------------------------------------------------//
    A     #sqSequencer.STEP.Jump;
    JCN   x021;

    R     #sqSequencer.STEP.Jump;
    R     #sqSequencer.STEP.Finished;

    L     11;     // Load next STEPNO to jump to if transition satisfied
    T     #sqSequencer.STEP.NumberNext; //Next Step11.

    JU    COMM;              // Transition satisfied, Exit, go to next step
x021: NOP   0;






    //============================= TRAN HEADER ==============================//
    // AUTOCODE   AUTOCODE   AUTOCODE   AUTOCODE   AUTOCODE   AUTOCODE   AUTO //
    // Bypass transition if manual jump:                                      //
    //------------------------------------------------------------------------//
    A     #sqSequencer.STEP.Finished;
    A     #smc.TRN_AND_JUMP;     //Manual jump is set Transition as bypassed
    JCN   COMM;              //exit

NETWORK
TITLE =S015::STEP 015:TRAN 022: Abort SIP
//----------------------------------------------------------------------------//
// TRAN   TRAN   TRAN   TRAN   TRAN   TRAN   TRAN   TRAN   TRAN   TRAN   TRAN //
// TRAN   TRAN   TRAN   TRAN   TRAN   TRAN   TRAN   TRAN   TRAN   TRAN   TRAN //
//----------------------------------------------------------------------------//
// Temperature has dropped 'NUM_SIP_ABORT' times.
//----------------------------------------------------------------------------//
// CONDITION   CONDITION   CONDITION   CONDITION   CONDITION   CONDITION   CO //
// CONDITION   CONDITION   CONDITION   CONDITION   CONDITION   CONDITION   CO //
//----------------------------------------------------------------------------//
//ABORT timer expired.
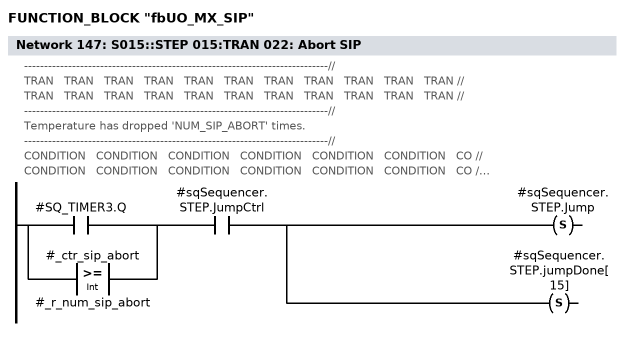
O #SQ_TIMER3.Q;
//Temperature has dropped NUM_SIP_ABORT times.
O(;
L 	#_ctr_sip_abort;
L 	#_r_num_sip_abort;
>=I;
);







    //============================= TRAN FOOTER ==============================//
    // Transition jump control:                                               //
    //------------------------------------------------------------------------//
    A     #sqSequencer.STEP.JumpCtrl;
    S     #sqSequencer.STEP.Jump;
    S     #sqSequencer.STEP.jumpDone[15];

NETWORK
TITLE =S015:t022::TRANS-v: EXIT TRANSITION AND READY THE NEXT STEP
    //------------------------------------------------------------------------//
    // Check the jump flag and jump to the next step if the transition        //
    // condition is true and has set the jump flag:                           //
    //------------------------------------------------------------------------//
    A     #sqSequencer.STEP.Jump;
    JCN   x022;

    R     #sqSequencer.STEP.Jump;
    R     #sqSequencer.STEP.Finished;

    L     17;     // Load next STEPNO to jump to if transition satisfied
    T     #sqSequencer.STEP.NumberNext; //Next Step17.

    JU    COMM;              // Transition satisfied, Exit, go to next step
x022: NOP   0;






NETWORK
TITLE =S015::STEP-015:EXIT TRANSITION:
    //========================== STEP TRANSFER ===============================//
    // Jump to the common step progression code:                              //
    //------------------------------------------------------------------------//
    JU    COMM;






NETWORK
TITLE =S016: STEP-16::UO_MX_SIP : MX complete
    //================================ STEP HEADER ===========================//
    // STEP016 STEP016 STEP016 STEP016
    // AUTOCODE   AUTOCODE   AUTOCODE   AUTOCODE   AUTOCODE   AUTOCODE   AUTO //
    // STEP016 STEP016 STEP016 STEP016
    //------------------------------------------------------------------------//
    // Log SIP completion time.
    // Clear pulse_counter.
    // Close Mx steam supply on WFI/PS.
    // Log all temperatures.
    //------------------------------------------------------------------------//
S016: NOP   0;

      SET;
      R     #sqSequencer.STEP.jumpDone[16];
      A     #sqSequencer.CMD.Pause; //If paused jump
      JC    COMM;

NETWORK
TITLE =S016:STEP-16:Begin Action

